# EPICS substitutions: db/ecmcEL2502.substitutions
file ecmcEL2502-chX.template
{
	pattern {CH_ID, LINR,    ESLO,            EOFF,    EGU,        PREC, LOW, LOLO, HIGH, HIHI, HYST, LLSV,       LSV,        HSV,        HHSV      }
		{1,     "SLOPE", 7.324442274E-4,  0,      "V",     0,    0,   0,    0,    0,    0,    "NO_ALARM", "NO_ALARM", "NO_ALARM", "NO_ALARM"}
		{2,     "SLOPE", 7.324442274E-4,  0,      "V",     0,    0,   0,    0,    0,    0,    "NO_ALARM", "NO_ALARM", "NO_ALARM", "NO_ALARM"}
}
